// Mitsubishi GX Works2 project: BookEX6_32 Shift_old   PLC: Q13UDV

// global labels: Global
VAR_GLOBAL
  bVar0 AT M5000 : BOOL;
  abArray0 AT M5010 : ARRAY [0..49] OF BOOL;
  sStr0 AT D5000 : STRING[199];
  sStr1 AT D5100 : STRING[199];
  sStr2 AT D5200 : STRING[199];
  sStr3 AT D5300 : STRING[199];
  sStr4 AT D5400 : STRING[199];
  sStr5 AT D5500 : STRING[199];
  sStr6 AT D5600 : STRING[199];
  sStr7 AT D5700 : STRING[199];
  sStr8 AT D5800 : STRING[199];
  sStr9 AT D5900 : STRING[199];
  iVar0 AT D4500 : INT;
  iVar1 AT D4501 : INT;
  iVar2 AT D4502 : INT;
  iVar3 AT D4503 : INT;
  iVar4 AT D4504 : INT;
  iVar5 AT D4505 : INT;
  iVar6 AT D4506 : INT;
  iVar7 AT D4507 : INT;
  iVar8 AT D4508 : INT;
  iVar9 AT D4509 : INT;
  dVar0 AT D4510 : DINT;
  dVar1 AT D4512 : DINT;
  dVar2 AT D4514 : DINT;
  dVar3 AT D4516 : DINT;
  dVar4 AT D4518 : DINT;
  dVar5 AT D4520 : DINT;
  dVar6 AT D4522 : DINT;
  dVar7 AT D4524 : DINT;
  dVar8 AT D4526 : DINT;
  dVar9 AT D4528 : DINT;
  wVar0 AT D4530 : WORD;
  wVar1 AT D4531 : WORD;
  wVar2 AT D4532 : WORD;
  wVar3 AT D4533 : WORD;
  wVar4 AT D4534 : WORD;
  wVar5 AT D4535 : WORD;
  wVar6 AT D4536 : WORD;
  wVar7 AT D4537 : WORD;
  wVar8 AT D4538 : WORD;
  wVar9 AT D4539 : WORD;
  dwVar0 AT D4540 : DWORD;
  dwVar1 AT D4542 : DWORD;
  dwVar2 AT D4544 : DWORD;
  dwVar3 AT D4546 : DWORD;
  dwVar4 AT D4548 : DWORD;
  dwVar5 AT D4550 : DWORD;
  dwVar6 AT D4552 : DWORD;
  dwVar7 AT D4554 : DWORD;
  dwVar8 AT D4556 : DWORD;
  dwVar9 AT D4558 : DWORD;
  fsVar0 AT D4560 : REAL;
  fsVar1 AT D4562 : REAL;
  fsVar2 AT D4564 : REAL;
  fsVar3 AT D4566 : REAL;
  fsVar4 AT D4568 : REAL;
  fsVar5 AT D4570 : REAL;
  fsVar6 AT D4572 : REAL;
  fsVar7 AT D4574 : REAL;
  fsVar8 AT D4576 : REAL;
  fsVar9 AT D4578 : REAL;
  fdVar0 AT D4580 : LREAL;
  tTime0 AT D4620 : TIME;
  tTime1 AT D4622 : TIME;
  tTime2 AT D4624 : TIME;
  tTime3 AT D4626 : TIME;
  tTime4 AT D4628 : TIME;
  tTime5 AT D4630 : TIME;
  tTime6 AT D4632 : TIME;
  tTime7 AT D4634 : TIME;
  tTime8 AT D4636 : TIME;
  tTime9 AT D4638 : TIME;
  tTime10 AT D4640 : TIME;
  bVar1 AT M5001 : BOOL;
  bVar2 AT M5002 : BOOL;
  bVar3 AT M5003 : BOOL;
  bVar4 AT M5004 : BOOL;
  bVar5 AT M5005 : BOOL;
  bVar6 AT M5006 : BOOL;
  bVar7 AT M5007 : BOOL;
  bVar8 AT M5008 : BOOL;
  bVar9 AT M5009 : BOOL;
  abArray1 AT M5060 : ARRAY [0..49] OF BOOL;
  abArray2 AT M5110 : ARRAY [0..49] OF BOOL;
  abArray3 AT M5160 : ARRAY [0..49] OF BOOL;
  abArray4 AT M5210 : ARRAY [0..49] OF BOOL;
  abArray5 AT M5260 : ARRAY [0..49] OF BOOL;
  abArray6 AT M5310 : ARRAY [0..49] OF BOOL;
  abArray7 AT M5360 : ARRAY [0..49] OF BOOL;
  abArray8 AT M5410 : ARRAY [0..49] OF BOOL;
  abArray9 AT M5460 : ARRAY [0..49] OF BOOL;
  fdVar1 AT D4584 : LREAL;
  fdVar2 AT D4588 : LREAL;
  fdVar3 AT D4592 : LREAL;
  fdVar4 AT D4596 : LREAL;
  fdVar5 AT D4600 : LREAL;
  fdVar6 AT D4604 : LREAL;
  fdVar7 AT D4608 : LREAL;
  fdVar8 AT D4612 : LREAL;
  fdVar9 AT D4616 : LREAL;
  afsPen0 AT D2000 : ARRAY [0..499] OF REAL;
  afsPen1 AT D3000 : ARRAY [0..499] OF REAL;
  adwD10 AT D10 : ARRAY [0..9] OF DWORD;
  awLeft AT D10 : ARRAY [0..9] OF WORD;
  awRight AT D20 : ARRAY [0..9] OF WORD;
  awBuffer AT D30 : ARRAY [0..59] OF WORD;
  awDigit AT D100 : ARRAY [0..11,0..9] OF WORD;
  abM10 AT M10 : ARRAY [0..19] OF BOOL;
END_VAR
// user libraries (not included): HMI

FUNCTION BitCount
VAR_INPUT
  w_IN : WORD;
END_VAR
VAR
  wTmp : WORD;
  iCnt : INT;
END_VAR
;
iCnt := 0;
wTmp := w_IN;
WHILE (wTmp AND HFFFF) <> 0 DO
	IF (wTmp  AND 1) <> 0 THEN iCnt := iCnt + 1; END_IF;
	SFR(TRUE, 1, wTmp);
END_WHILE;
BitCount := iCnt;
END_FUNCTION

FUNCTION BitLoadPos
VAR_INPUT
  w_IN : WORD;
END_VAR
VAR
  wInput : WORD;
END_VAR
VAR_INPUT
  b_Val : BOOL;
  i_Pos : INT;
END_VAR
VAR
  wTmp1 : WORD;
  wTmp2 : WORD;
END_VAR
;
wTmp1 := H0001;
wInput := w_IN;
IF b_Val THEN
	SFL(TRUE, i_Pos, wTmp1);
	wTmp2 := wInput OR wTmp1;
ELSE
	SFL(TRUE, i_Pos, wTmp1);
	wTmp2 := wInput AND NOT wTmp1;
END_IF;
BitLoadPos := wTmp2;
END_FUNCTION

FUNCTION BitReset
VAR_INPUT
  w_IN : WORD;
END_VAR
VAR
  wInput : WORD;
END_VAR
VAR_INPUT
  i_Pos : INT;
END_VAR
VAR
  wTmp1 : WORD;
  wTmp2 : WORD;
END_VAR
;
wTmp1 := H0001;
wInput := w_IN;
SFL(TRUE, i_Pos, wTmp1);
wTmp2 := wInput AND NOT wTmp1;
BitReset := wTmp2;
END_FUNCTION

FUNCTION BitSet
VAR_INPUT
  w_IN : WORD;
END_VAR
VAR
  wInput : WORD;
END_VAR
VAR_INPUT
  i_Pos : INT;
END_VAR
VAR
  wTmp1 : WORD;
  wTmp2 : WORD;
END_VAR
;
wTmp1 := H0001;
wInput := w_IN;
SFL(TRUE, i_Pos, wTmp1);
wTmp2 := wInput OR wTmp1;
BitSet := wTmp2;
END_FUNCTION

FUNCTION BitToggle
VAR_INPUT
  w_IN : WORD;
  i_Pos : INT;
END_VAR
VAR
  wInput : WORD;
  wTmp1 : WORD;
  wTmp2 : WORD;
END_VAR
;
wTmp1 := H0001;
wInput := w_IN;
SFL(TRUE, i_Pos, wTmp1);
wTmp2 := wInput XOR wTmp1;
BitToggle := wTmp2;
END_FUNCTION

FUNCTION_BLOCK EBIncDec
VAR_INPUT
  i_Old : INT;
END_VAR
VAR_OUTPUT
  b_ChgUp : BOOL;
END_VAR
VAR_INPUT
  b_Inc : BOOL;
END_VAR
VAR
  ix : INT;
END_VAR
VAR_OUTPUT
  i_New : INT;
END_VAR
VAR_INPUT
  b_Dec : BOOL;
END_VAR
VAR_OUTPUT
  b_ChgDw : BOOL;
END_VAR
;
IF NOT b_Inc AND NOT b_Dec THEN
	RETURN;
END_IF;
IF b_Inc THEN
	IF  (i_Old = 9) OR (i_Old = 0) THEN
		b_ChgUp := FALSE;
	ELSE
		i_New := i_Old + 1;
		b_ChgUp := TRUE;
		FOR ix := 0 TO 9 DO 
			awBuffer[ix+20] := awDigit[10, ix];
			awBuffer[ix+50] := awDigit[i_New, ix];
		END_FOR;
	END_IF;
ELSIF b_Dec THEN
	IF  (i_Old = 1) OR (i_Old = 0) THEN
		b_ChgDw := FALSE;
	ELSE
		i_New := i_Old - 1;
		b_ChgDw := TRUE;
		FOR ix := 0 TO 9 DO 
			awBuffer[ix+0] := awDigit[11, ix];
			awBuffer[ix+30] := awDigit[i_New, ix];
		END_FOR;
	END_IF;
END_IF;
END_FUNCTION_BLOCK

FUNCTION_BLOCK EBScroll
VAR_INPUT
  b_EN : BOOL;
  b_Up : BOOL;
  b_Dw : BOOL;
END_VAR
VAR_OUTPUT
  b_Ing : BOOL;
  b_Comp : BOOL;
END_VAR
VAR
  ix : INT;
  iCnt : INT;
END_VAR
VAR_IN_OUT
  i_Old : INT;
  i_New : INT;
END_VAR
VAR
  fbTimer : TON;
END_VAR
;
IF NOT b_EN THEN
	iCnt := 0;
	b_Ing := FALSE;
	b_Comp := FALSE;
	fbTimer(IN:=FALSE);
	RETURN;
END_IF;

IF b_Up THEN
	CASE iCnt OF 
		0 : 	FOR ix := 0 TO 9 DO 
					awBuffer[ix+10] := 0;
					awBuffer[ix+40] := awDigit[i_Old, ix];
				END_FOR;
				b_Comp := FALSE;
				b_Ing := TRUE;
				iCnt := iCnt + 1;
		1..10 : 
				fbTimer(IN := TRUE , PT:=T#500ms);
				IF fbTimer.Q THEN
					fbTimer(IN:=FALSE);
					iCnt := iCnt+1;
					SFTWR(TRUE, 30, 1, awBuffer[0] );
					SFTWR(TRUE, 30, 1, awBuffer[30] );
				END_IF;
		11..14 : 
				fbTimer(IN := TRUE , PT:=T#500ms);
				IF fbTimer.Q THEN
					fbTimer(IN:=FALSE);
					iCnt := iCnt+1;
					SFTWR(TRUE, 30, 1, awBuffer[0] );
				END_IF;
		15 :		
				b_Comp := TRUE;
				i_Old := i_New;
				b_Ing := FALSE;
				iCnt := 0;
	END_CASE;
ELSIF b_Dw THEN
	CASE iCnt OF 
		0 : 	FOR ix := 0 TO 9 DO 
					awBuffer[ix+10] := 0;
					awBuffer[ix+40] := awDigit[i_Old, ix];
				END_FOR;
				b_Comp := FALSE;
				b_Ing := TRUE;
				iCnt := iCnt + 1;
		1..10 : 
				fbTimer(IN := TRUE , PT:=T#500ms);
				IF fbTimer.Q THEN
					fbTimer(IN:=FALSE);
					iCnt := iCnt+1;
					SFTWL(TRUE, 30, 1, awBuffer[0] );
					SFTWL(TRUE, 30, 1, awBuffer[30] );
				END_IF;
		11..15 : 
				fbTimer(IN := TRUE , PT:=T#500ms);
				IF fbTimer.Q THEN
					fbTimer(IN:=FALSE);
					iCnt := iCnt+1;
					SFTWL(TRUE, 30, 1, awBuffer[0] );
				END_IF;
		16 :		
				b_Comp := TRUE;
				i_Old := i_New;
				b_Ing := FALSE;
				iCnt := 0;
	END_CASE;	
ELSE
	iCnt := 0;
	b_Ing := FALSE;
	b_Comp := FALSE;
	FOR ix := 0 TO 9 DO 
		awBuffer[ix+10] := 0;
		awBuffer[ix+40] := awDigit[i_Old, ix];
	END_FOR;
END_IF;

FOR ix := 0 TO 9 DO 
		awLeft[ix] := awBuffer[ix+10];
		awRight[ix] := awBuffer[ix+40];
END_FOR;
END_FUNCTION_BLOCK

FUNCTION_BLOCK EBScroll2
VAR_INPUT
  b_EN : BOOL;
  b_Up : BOOL;
  b_Dw : BOOL;
END_VAR
VAR_OUTPUT
  b_Ing : BOOL;
  b_Comp : BOOL;
END_VAR
VAR
  ix : INT;
  iCnt : INT;
END_VAR
VAR_IN_OUT
  i_Old : INT;
  i_New : INT;
END_VAR
VAR
  fbTimer : TON;
  dwTemp1 : DWORD;
  dwTemp2 : DWORD;
  dwTemp3 : DWORD;
  dwTemp4 : DWORD;
  dwTemp5 : DWORD;
  iy : INT;
END_VAR
;
IF NOT b_EN THEN
	iCnt := 0;
	b_Ing := FALSE;
	b_Comp := FALSE;
	fbTimer(IN:=FALSE);
	RETURN;
END_IF;

IF b_Up THEN
	CASE iCnt OF 
		0 : 	FOR ix := 0 TO 9 DO 
					awBuffer[ix+10] := 0;
					awBuffer[ix+40] := awDigit[i_Old, ix];
				END_FOR;
				b_Comp := FALSE;
				b_Ing := TRUE;
				iCnt := iCnt + 1;
		1..16 : 
				fbTimer(IN := TRUE , PT:=T#500ms);
				IF fbTimer.Q THEN
					fbTimer(IN:=FALSE);
					iCnt := iCnt+1;
					FOR iy := 0 TO 9 DO
						dwTemp1 			:= WORD_TO_DWORD(awBuffer[iy+40]) AND H000000FF;
						dwTemp2 			:= SHL( WORD_TO_DWORD(awBuffer[iy+10]), 8) AND H0000FF00;
						dwTemp3 			:= SHL( WORD_TO_DWORD(awBuffer[iy+50]), 16) AND H00FF0000;
						dwTemp4 			:= SHL( WORD_TO_DWORD(awBuffer[iy+20]), 24) AND HFF000000;
						dwTemp5 			:= dwTemp1 OR dwTemp2 OR dwTemp3 OR dwTemp4;
						dwTemp5 			:= SHR(dwTemp5, 1);
						awBuffer[iy+40] 	:= DWORD_TO_WORD(dwTemp5 AND H000000FF);
						awBuffer[iy+10] 	:= DWORD_TO_WORD(SHR(dwTemp5, 8) AND H000000FF);
						awBuffer[iy+50] 	:= DWORD_TO_WORD(SHR(dwTemp5, 16) AND H000000FF);
						awBuffer[iy+20]	:= DWORD_TO_WORD(SHR(dwTemp5, 24) AND H000000FF);
					END_FOR;
				END_IF;
		17 :		
				b_Comp := TRUE;
				i_Old := i_New;
				b_Ing := FALSE;
				iCnt := 0;
	END_CASE;
ELSIF b_Dw THEN
	CASE iCnt OF 
		0 : 	FOR ix := 0 TO 9 DO 
					awBuffer[ix+10] := 0;
					awBuffer[ix+40] := awDigit[i_Old, ix];
				END_FOR;
				b_Comp := FALSE;
				b_Ing := TRUE;
				iCnt := iCnt + 1;
		1..16 : 
				fbTimer(IN := TRUE , PT:=T#500ms);
				IF fbTimer.Q THEN
					fbTimer(IN:=FALSE);
					iCnt := iCnt+1;
					FOR iy := 0 TO 9 DO
						dwTemp1 			:= WORD_TO_DWORD(awBuffer[iy+30]) AND H000000FF;
						dwTemp2 			:= SHL( WORD_TO_DWORD(awBuffer[iy]), 8) AND H0000FF00;
						dwTemp3 			:= SHL( WORD_TO_DWORD(awBuffer[iy+40]), 16) AND H00FF0000;
						dwTemp4 			:= SHL( WORD_TO_DWORD(awBuffer[iy+10]), 24) AND HFF000000;
						dwTemp5 			:= dwTemp1 OR dwTemp2 OR dwTemp3 OR dwTemp4;
						dwTemp5 			:= SHL(dwTemp5, 1);
						awBuffer[iy+30] 	:= DWORD_TO_WORD(dwTemp5 AND H000000FF);
						awBuffer[iy] 		:= DWORD_TO_WORD(SHR(dwTemp5, 8) AND H000000FF);
						awBuffer[iy+40] 	:= DWORD_TO_WORD(SHR(dwTemp5, 16) AND H000000FF);
						awBuffer[iy+10]	:= DWORD_TO_WORD(SHR(dwTemp5, 24) AND H000000FF);
					END_FOR;
				END_IF;
		17 :		
				b_Comp := TRUE;
				i_Old := i_New;
				b_Ing := FALSE;
				iCnt := 0;
	END_CASE;	
ELSE
	iCnt := 0;
	b_Ing := FALSE;
	b_Comp := FALSE;
	FOR ix := 0 TO 9 DO 
		awBuffer[ix+10] := 0;
		awBuffer[ix+40] := awDigit[i_Old, ix];
	END_FOR;
END_IF;

FOR ix := 0 TO 9 DO 
		awLeft[ix] := awBuffer[ix+10];
		awRight[ix] := awBuffer[ix+40];
END_FOR;
END_FUNCTION_BLOCK

PROGRAM ExBSFR
(* structured ladder/FBD written out as ST: instructions are called as NAME(EN, inputs, outputs); _pN, _eN, _tN stand for wires *)
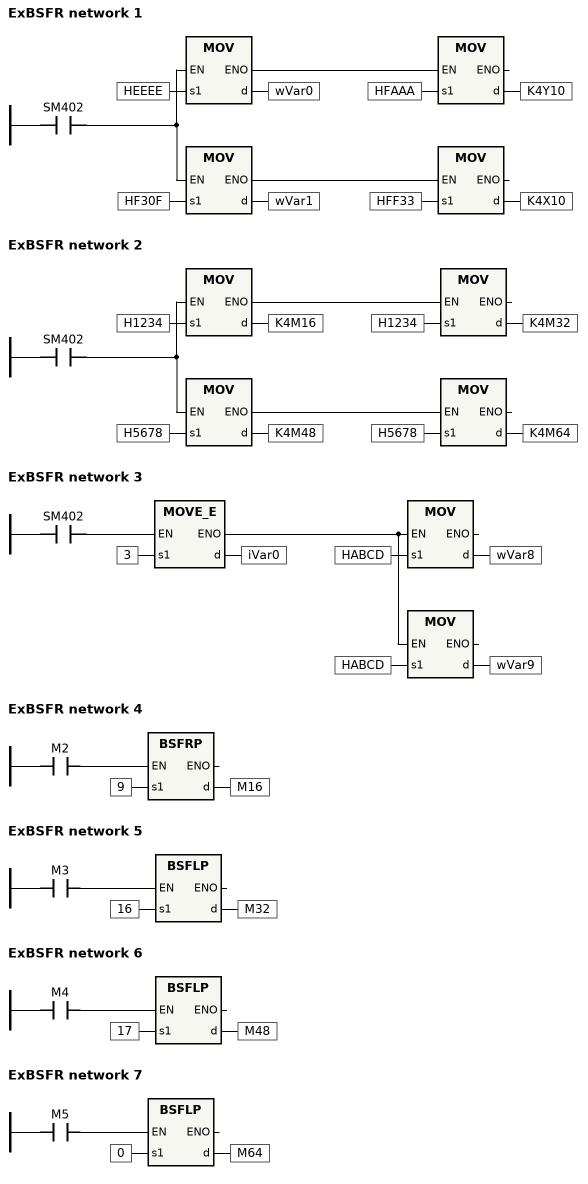
(* network 1 *)
_e1 := MOV(SM402, HEEEE, wVar0);
MOV(_e1, HFAAA, K4Y10);
_e2 := MOV(SM402, HF30F, wVar1);
MOV(_e2, HFF33, K4X10);
(* network 2 *)
_e1 := MOV(SM402, H1234, K4M16);
MOV(_e1, H1234, K4M32);
_e2 := MOV(SM402, H5678, K4M48);
MOV(_e2, H5678, K4M64);
(* network 3 *)
_e1 := MOVE_E(SM402, 3, iVar0);
MOV(_e1, HABCD, wVar8);
MOV(_e1, HABCD, wVar9);
(* network 4 *)
BSFRP(M2, 9, M16);
(* network 5 *)
BSFLP(M3, 16, M32);
(* network 6 *)
BSFLP(M4, 17, M48);
(* network 7 *)
BSFLP(M5, 0, M64);
END_PROGRAM

PROGRAM ExDisplay
VAR
  Mov8WORD_1 : Mov8WORD;
  Mov8WORD_2 : Mov8WORD;
  Mov8WORD_3 : Mov8WORD;
  Mov8WORD_4 : Mov8WORD;
  Mov8WORD_5 : Mov8WORD;
  Mov8WORD_6 : Mov8WORD;
  Mov8WORD_7 : Mov8WORD;
  Mov8WORD_8 : Mov8WORD;
  Mov8WORD_9 : Mov8WORD;
  Mov8WORD_10 : Mov8WORD;
  Mov8WORD_11 : Mov8WORD;
  Mov8WORD_12 : Mov8WORD;
  Mov8WORD_13 : Mov8WORD;
  Mov8WORD_14 : Mov8WORD;
  Mov8WORD_15 : Mov8WORD;
  OldIdx : INT;
  NewIdx : INT;
  bDwFlag : BOOL;
  bUpFlag : BOOL;
  EBScroll_1 : EBScroll;
  bScroll : BOOL;
  bStop : BOOL;
  EBIncDec_1 : EBIncDec;
END_VAR
(* structured ladder/FBD written out as ST: instructions are called as NAME(EN, inputs, outputs); _pN, _eN, _tN stand for wires *)
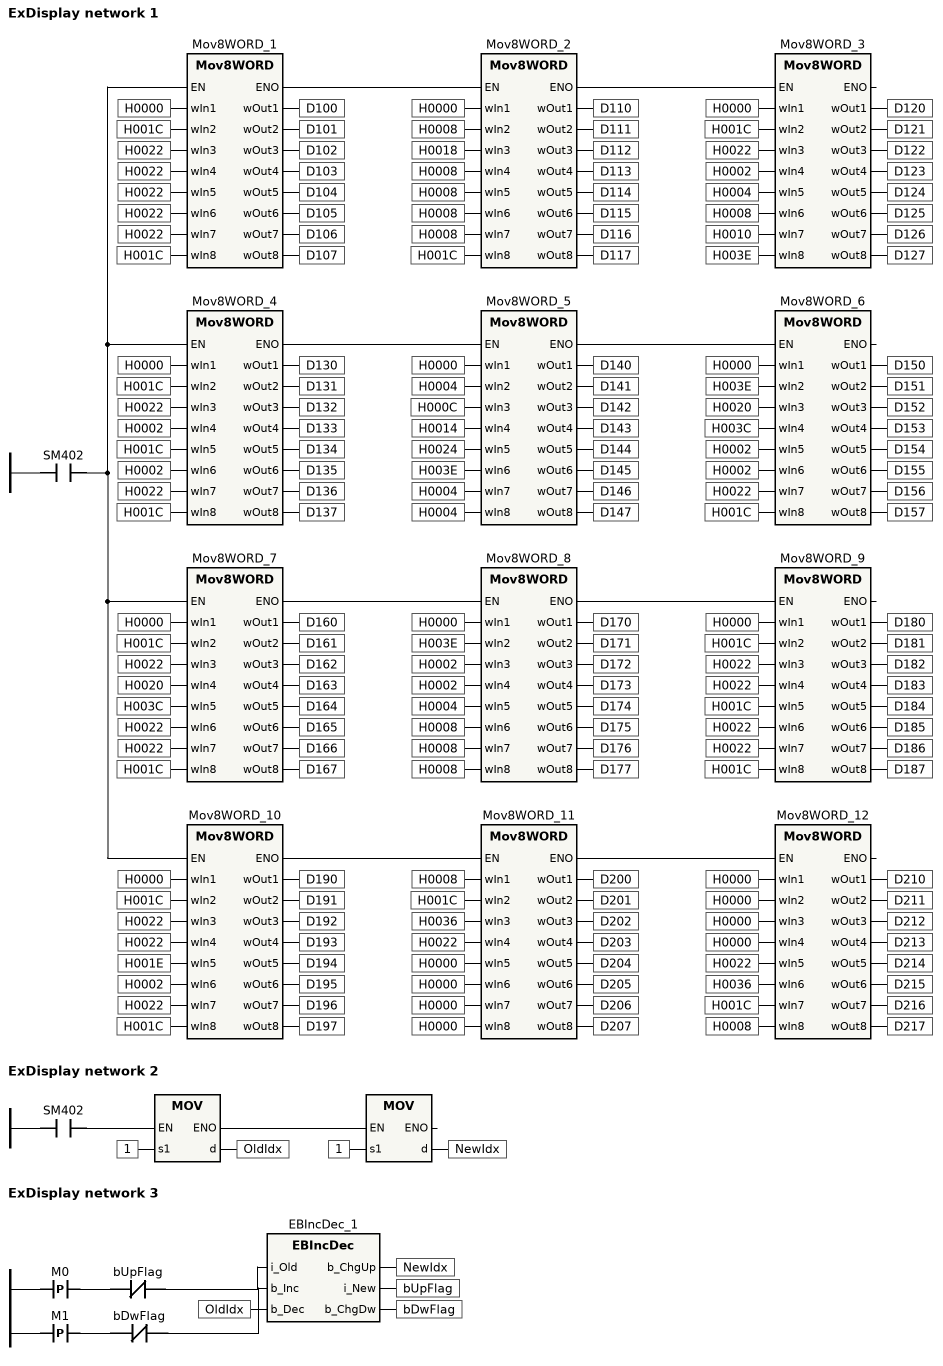
(* network 1 *)
Mov8WORD_1(EN := SM402, wIn1 := H0000, wIn2 := H001C, wIn3 := H0022, wIn4 := H0022, wIn5 := H0022, wIn6 := H0022, wIn7 := H0022, wIn8 := H001C, wOut1 => D100, wOut2 => D101, wOut3 => D102, wOut4 => D103, wOut5 => D104, wOut6 => D105, wOut7 => D106, wOut8 => D107);
Mov8WORD_2(EN := Mov8WORD_1.ENO, wIn1 := H0000, wIn2 := H0008, wIn3 := H0018, wIn4 := H0008, wIn5 := H0008, wIn6 := H0008, wIn7 := H0008, wIn8 := H001C, wOut1 => D110, wOut2 => D111, wOut3 => D112, wOut4 => D113, wOut5 => D114, wOut6 => D115, wOut7 => D116, wOut8 => D117);
Mov8WORD_3(EN := Mov8WORD_2.ENO, wIn1 := H0000, wIn2 := H001C, wIn3 := H0022, wIn4 := H0002, wIn5 := H0004, wIn6 := H0008, wIn7 := H0010, wIn8 := H003E, wOut1 => D120, wOut2 => D121, wOut3 => D122, wOut4 => D123, wOut5 => D124, wOut6 => D125, wOut7 => D126, wOut8 => D127);
Mov8WORD_4(EN := SM402, wIn1 := H0000, wIn2 := H001C, wIn3 := H0022, wIn4 := H0002, wIn5 := H001C, wIn6 := H0002, wIn7 := H0022, wIn8 := H001C, wOut1 => D130, wOut2 => D131, wOut3 => D132, wOut4 => D133, wOut5 => D134, wOut6 => D135, wOut7 => D136, wOut8 => D137);
Mov8WORD_5(EN := Mov8WORD_4.ENO, wIn1 := H0000, wIn2 := H0004, wIn3 := H000C, wIn4 := H0014, wIn5 := H0024, wIn6 := H003E, wIn7 := H0004, wIn8 := H0004, wOut1 => D140, wOut2 => D141, wOut3 => D142, wOut4 => D143, wOut5 => D144, wOut6 => D145, wOut7 => D146, wOut8 => D147);
Mov8WORD_6(EN := Mov8WORD_5.ENO, wIn1 := H0000, wIn2 := H003E, wIn3 := H0020, wIn4 := H003C, wIn5 := H0002, wIn6 := H0002, wIn7 := H0022, wIn8 := H001C, wOut1 => D150, wOut2 => D151, wOut3 => D152, wOut4 => D153, wOut5 => D154, wOut6 => D155, wOut7 => D156, wOut8 => D157);
Mov8WORD_7(EN := SM402, wIn1 := H0000, wIn2 := H001C, wIn3 := H0022, wIn4 := H0020, wIn5 := H003C, wIn6 := H0022, wIn7 := H0022, wIn8 := H001C, wOut1 => D160, wOut2 => D161, wOut3 => D162, wOut4 => D163, wOut5 => D164, wOut6 => D165, wOut7 => D166, wOut8 => D167);
Mov8WORD_8(EN := Mov8WORD_7.ENO, wIn1 := H0000, wIn2 := H003E, wIn3 := H0002, wIn4 := H0002, wIn5 := H0004, wIn6 := H0008, wIn7 := H0008, wIn8 := H0008, wOut1 => D170, wOut2 => D171, wOut3 => D172, wOut4 => D173, wOut5 => D174, wOut6 => D175, wOut7 => D176, wOut8 => D177);
Mov8WORD_9(EN := Mov8WORD_8.ENO, wIn1 := H0000, wIn2 := H001C, wIn3 := H0022, wIn4 := H0022, wIn5 := H001C, wIn6 := H0022, wIn7 := H0022, wIn8 := H001C, wOut1 => D180, wOut2 => D181, wOut3 => D182, wOut4 => D183, wOut5 => D184, wOut6 => D185, wOut7 => D186, wOut8 => D187);
Mov8WORD_10(EN := SM402, wIn1 := H0000, wIn2 := H001C, wIn3 := H0022, wIn4 := H0022, wIn5 := H001E, wIn6 := H0002, wIn7 := H0022, wIn8 := H001C, wOut1 => D190, wOut2 => D191, wOut3 => D192, wOut4 => D193, wOut5 => D194, wOut6 => D195, wOut7 => D196, wOut8 => D197);
Mov8WORD_11(EN := Mov8WORD_10.ENO, wIn1 := H0008, wIn2 := H001C, wIn3 := H0036, wIn4 := H0022, wIn5 := H0000, wIn6 := H0000, wIn7 := H0000, wIn8 := H0000, wOut1 => D200, wOut2 => D201, wOut3 => D202, wOut4 => D203, wOut5 => D204, wOut6 => D205, wOut7 => D206, wOut8 => D207);
Mov8WORD_12(EN := Mov8WORD_11.ENO, wIn1 := H0000, wIn2 := H0000, wIn3 := H0000, wIn4 := H0000, wIn5 := H0022, wIn6 := H0036, wIn7 := H001C, wIn8 := H0008, wOut1 => D210, wOut2 => D211, wOut3 => D212, wOut4 => D213, wOut5 => D214, wOut6 => D215, wOut7 => D216, wOut8 => D217);
(* network 2 *)
_e1 := MOV(SM402, 1, OldIdx);
MOV(_e1, 1, NewIdx);
(* network 3 *)
EBIncDec_1(i_Old := LDP(TRUE, M0) AND NOT bUpFlag, b_Inc := LDP(TRUE, M1) AND NOT bDwFlag, b_Dec := OldIdx, b_ChgUp => NewIdx, i_New => bUpFlag, b_ChgDw => bDwFlag);
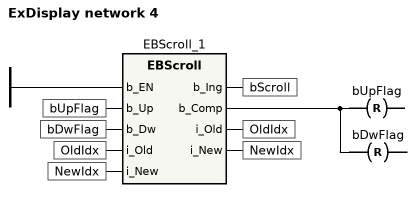
(* network 4 *)
EBScroll_1(b_EN := TRUE, b_Up := bUpFlag, b_Dw := bDwFlag, i_Old := OldIdx, i_New := NewIdx, b_Ing => bScroll);
RST(EBScroll_1.b_Comp, bUpFlag);
OldIdx := EBScroll_1.i_Old;
RST(EBScroll_1.b_Comp, bDwFlag);
NewIdx := EBScroll_1.i_New;
END_PROGRAM

PROGRAM ExDisplay2
VAR
  Mov8WORD_1 : Mov8WORD;
  Mov8WORD_2 : Mov8WORD;
  Mov8WORD_3 : Mov8WORD;
  Mov8WORD_4 : Mov8WORD;
  Mov8WORD_5 : Mov8WORD;
  Mov8WORD_6 : Mov8WORD;
  Mov8WORD_7 : Mov8WORD;
  Mov8WORD_8 : Mov8WORD;
  Mov8WORD_9 : Mov8WORD;
  Mov8WORD_10 : Mov8WORD;
  Mov8WORD_11 : Mov8WORD;
  Mov8WORD_12 : Mov8WORD;
  Mov8WORD_13 : Mov8WORD;
  Mov8WORD_14 : Mov8WORD;
  Mov8WORD_15 : Mov8WORD;
  OldIdx : INT;
  NewIdx : INT;
  bDwFlag : BOOL;
  bUpFlag : BOOL;
  bScroll : BOOL;
  bStop : BOOL;
  EBScroll_1 : EBScroll2;
  EBIncDec_1 : EBIncDec;
END_VAR
(* structured ladder/FBD written out as ST: instructions are called as NAME(EN, inputs, outputs); _pN, _eN, _tN stand for wires *)
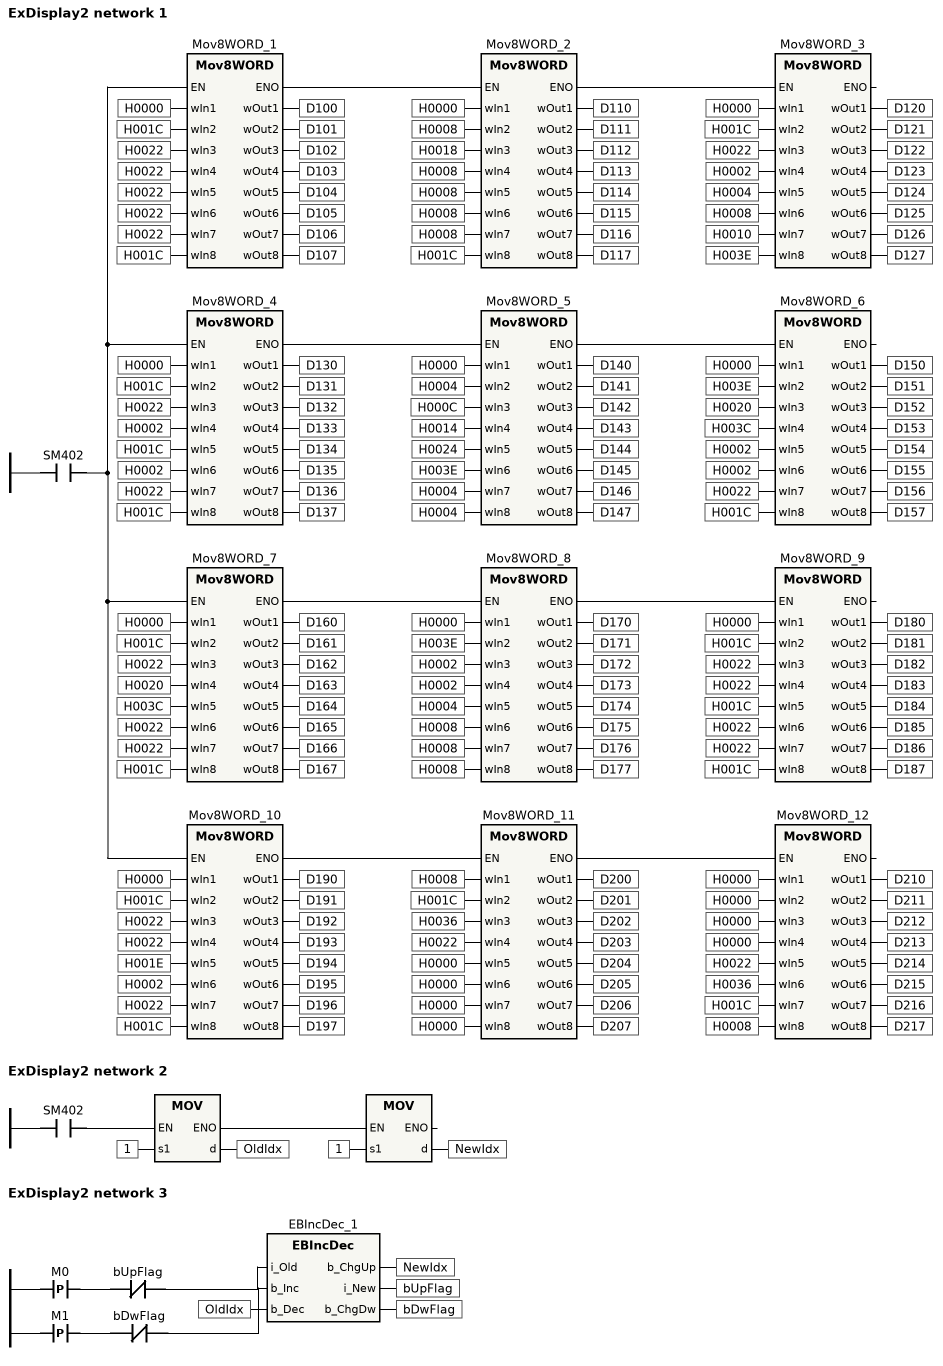
(* network 1 *)
Mov8WORD_1(EN := SM402, wIn1 := H0000, wIn2 := H001C, wIn3 := H0022, wIn4 := H0022, wIn5 := H0022, wIn6 := H0022, wIn7 := H0022, wIn8 := H001C, wOut1 => D100, wOut2 => D101, wOut3 => D102, wOut4 => D103, wOut5 => D104, wOut6 => D105, wOut7 => D106, wOut8 => D107);
Mov8WORD_2(EN := Mov8WORD_1.ENO, wIn1 := H0000, wIn2 := H0008, wIn3 := H0018, wIn4 := H0008, wIn5 := H0008, wIn6 := H0008, wIn7 := H0008, wIn8 := H001C, wOut1 => D110, wOut2 => D111, wOut3 => D112, wOut4 => D113, wOut5 => D114, wOut6 => D115, wOut7 => D116, wOut8 => D117);
Mov8WORD_3(EN := Mov8WORD_2.ENO, wIn1 := H0000, wIn2 := H001C, wIn3 := H0022, wIn4 := H0002, wIn5 := H0004, wIn6 := H0008, wIn7 := H0010, wIn8 := H003E, wOut1 => D120, wOut2 => D121, wOut3 => D122, wOut4 => D123, wOut5 => D124, wOut6 => D125, wOut7 => D126, wOut8 => D127);
Mov8WORD_4(EN := SM402, wIn1 := H0000, wIn2 := H001C, wIn3 := H0022, wIn4 := H0002, wIn5 := H001C, wIn6 := H0002, wIn7 := H0022, wIn8 := H001C, wOut1 => D130, wOut2 => D131, wOut3 => D132, wOut4 => D133, wOut5 => D134, wOut6 => D135, wOut7 => D136, wOut8 => D137);
Mov8WORD_5(EN := Mov8WORD_4.ENO, wIn1 := H0000, wIn2 := H0004, wIn3 := H000C, wIn4 := H0014, wIn5 := H0024, wIn6 := H003E, wIn7 := H0004, wIn8 := H0004, wOut1 => D140, wOut2 => D141, wOut3 => D142, wOut4 => D143, wOut5 => D144, wOut6 => D145, wOut7 => D146, wOut8 => D147);
Mov8WORD_6(EN := Mov8WORD_5.ENO, wIn1 := H0000, wIn2 := H003E, wIn3 := H0020, wIn4 := H003C, wIn5 := H0002, wIn6 := H0002, wIn7 := H0022, wIn8 := H001C, wOut1 => D150, wOut2 => D151, wOut3 => D152, wOut4 => D153, wOut5 => D154, wOut6 => D155, wOut7 => D156, wOut8 => D157);
Mov8WORD_7(EN := SM402, wIn1 := H0000, wIn2 := H001C, wIn3 := H0022, wIn4 := H0020, wIn5 := H003C, wIn6 := H0022, wIn7 := H0022, wIn8 := H001C, wOut1 => D160, wOut2 => D161, wOut3 => D162, wOut4 => D163, wOut5 => D164, wOut6 => D165, wOut7 => D166, wOut8 => D167);
Mov8WORD_8(EN := Mov8WORD_7.ENO, wIn1 := H0000, wIn2 := H003E, wIn3 := H0002, wIn4 := H0002, wIn5 := H0004, wIn6 := H0008, wIn7 := H0008, wIn8 := H0008, wOut1 => D170, wOut2 => D171, wOut3 => D172, wOut4 => D173, wOut5 => D174, wOut6 => D175, wOut7 => D176, wOut8 => D177);
Mov8WORD_9(EN := Mov8WORD_8.ENO, wIn1 := H0000, wIn2 := H001C, wIn3 := H0022, wIn4 := H0022, wIn5 := H001C, wIn6 := H0022, wIn7 := H0022, wIn8 := H001C, wOut1 => D180, wOut2 => D181, wOut3 => D182, wOut4 => D183, wOut5 => D184, wOut6 => D185, wOut7 => D186, wOut8 => D187);
Mov8WORD_10(EN := SM402, wIn1 := H0000, wIn2 := H001C, wIn3 := H0022, wIn4 := H0022, wIn5 := H001E, wIn6 := H0002, wIn7 := H0022, wIn8 := H001C, wOut1 => D190, wOut2 => D191, wOut3 => D192, wOut4 => D193, wOut5 => D194, wOut6 => D195, wOut7 => D196, wOut8 => D197);
Mov8WORD_11(EN := Mov8WORD_10.ENO, wIn1 := H0008, wIn2 := H001C, wIn3 := H0036, wIn4 := H0022, wIn5 := H0000, wIn6 := H0000, wIn7 := H0000, wIn8 := H0000, wOut1 => D200, wOut2 => D201, wOut3 => D202, wOut4 => D203, wOut5 => D204, wOut6 => D205, wOut7 => D206, wOut8 => D207);
Mov8WORD_12(EN := Mov8WORD_11.ENO, wIn1 := H0000, wIn2 := H0000, wIn3 := H0000, wIn4 := H0000, wIn5 := H0022, wIn6 := H0036, wIn7 := H001C, wIn8 := H0008, wOut1 => D210, wOut2 => D211, wOut3 => D212, wOut4 => D213, wOut5 => D214, wOut6 => D215, wOut7 => D216, wOut8 => D217);
(* network 2 *)
_e1 := MOV(SM402, 1, OldIdx);
MOV(_e1, 1, NewIdx);
(* network 3 *)
EBIncDec_1(i_Old := LDP(TRUE, M0) AND NOT bUpFlag, b_Inc := LDP(TRUE, M1) AND NOT bDwFlag, b_Dec := OldIdx, b_ChgUp => NewIdx, i_New => bUpFlag, b_ChgDw => bDwFlag);
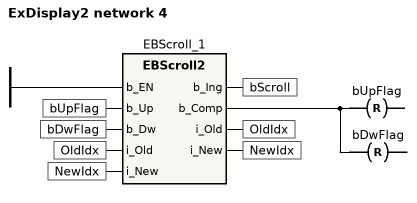
(* network 4 *)
EBScroll_1(b_EN := TRUE, b_Up := bUpFlag, b_Dw := bDwFlag, i_Old := OldIdx, i_New := NewIdx, b_Ing => bScroll);
RST(EBScroll_1.b_Comp, bUpFlag);
OldIdx := EBScroll_1.i_Old;
RST(EBScroll_1.b_Comp, bDwFlag);
NewIdx := EBScroll_1.i_New;
END_PROGRAM

PROGRAM ExDSFR
VAR
  Mov4WORD_1 : Mov4WORD;
  Mov8INT_1 : Mov8INT;
  Mov8INT_2 : Mov8INT;
END_VAR
(* structured ladder/FBD written out as ST: instructions are called as NAME(EN, inputs, outputs); _pN, _eN, _tN stand for wires *)
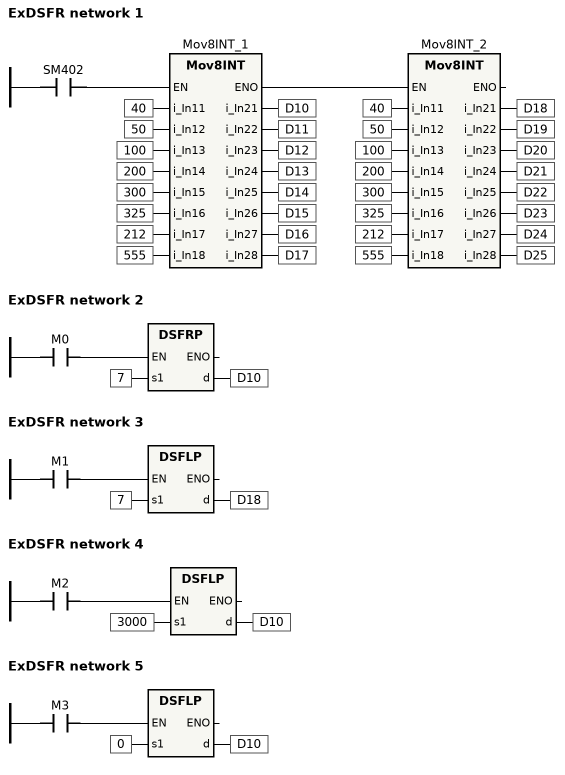
(* network 1 *)
Mov8INT_1(EN := SM402, i_In11 := 40, i_In12 := 50, i_In13 := 100, i_In14 := 200, i_In15 := 300, i_In16 := 325, i_In17 := 212, i_In18 := 555, i_In21 => D10, i_In22 => D11, i_In23 => D12, i_In24 => D13, i_In25 => D14, i_In26 => D15, i_In27 => D16, i_In28 => D17);
Mov8INT_2(EN := Mov8INT_1.ENO, i_In11 := 40, i_In12 := 50, i_In13 := 100, i_In14 := 200, i_In15 := 300, i_In16 := 325, i_In17 := 212, i_In18 := 555, i_In21 => D18, i_In22 => D19, i_In23 => D20, i_In24 => D21, i_In25 => D22, i_In26 => D23, i_In27 => D24, i_In28 => D25);
(* network 2 *)
DSFRP(M0, 7, D10);
(* network 3 *)
DSFLP(M1, 7, D18);
(* network 4 *)
DSFLP(M2, 3000, D10);
(* network 5 *)
DSFLP(M3, 0, D10);
END_PROGRAM

PROGRAM ExLib
(* structured ladder/FBD written out as ST: instructions are called as NAME(EN, inputs, outputs); _pN, _eN, _tN stand for wires *)
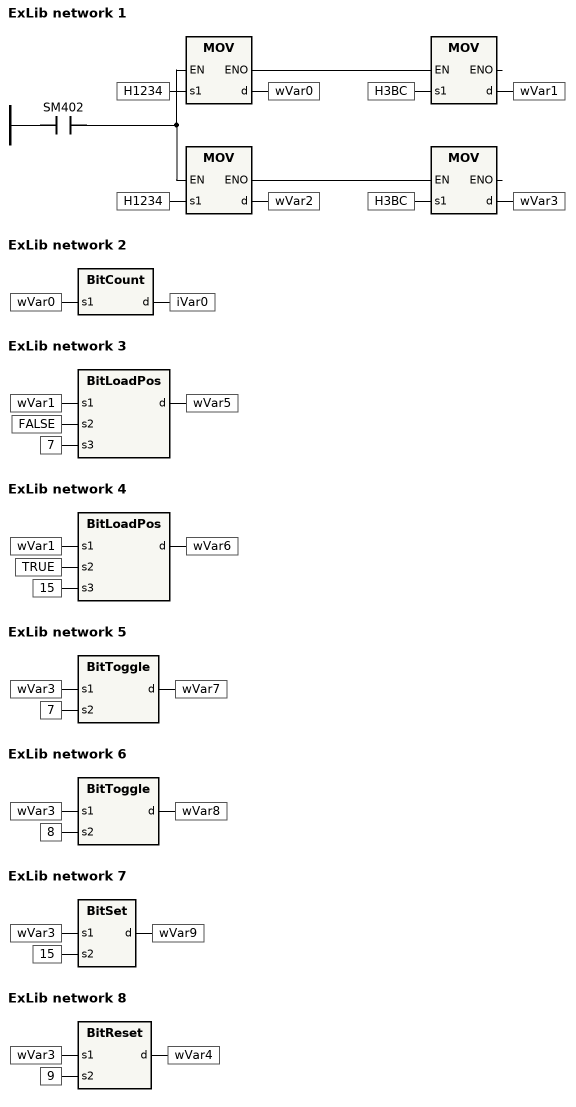
(* network 1 *)
_e1 := MOV(SM402, H1234, wVar0);
MOV(_e1, H3BC, wVar1);
_e2 := MOV(SM402, H1234, wVar2);
MOV(_e2, H3BC, wVar3);
(* network 2 *)
iVar0 := BitCount(wVar0);
(* network 3 *)
wVar5 := BitLoadPos(wVar1, FALSE, 7);
(* network 4 *)
wVar6 := BitLoadPos(wVar1, TRUE, 15);
(* network 5 *)
wVar7 := BitToggle(wVar3, 7);
(* network 6 *)
wVar8 := BitToggle(wVar3, 8);
(* network 7 *)
wVar9 := BitSet(wVar3, 15);
(* network 8 *)
wVar4 := BitReset(wVar3, 9);
END_PROGRAM

PROGRAM ExSFR
(* structured ladder/FBD written out as ST: instructions are called as NAME(EN, inputs, outputs); _pN, _eN, _tN stand for wires *)
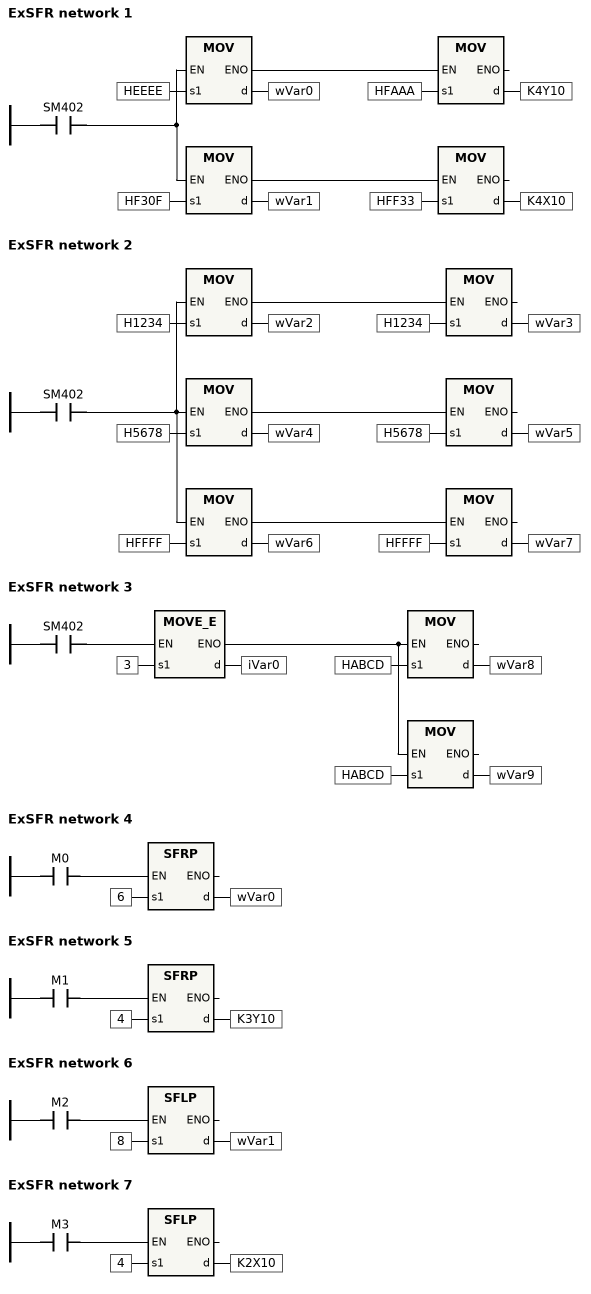
(* network 1 *)
_e1 := MOV(SM402, HEEEE, wVar0);
MOV(_e1, HFAAA, K4Y10);
_e2 := MOV(SM402, HF30F, wVar1);
MOV(_e2, HFF33, K4X10);
(* network 2 *)
_e1 := MOV(SM402, H1234, wVar2);
MOV(_e1, H1234, wVar3);
_e2 := MOV(SM402, H5678, wVar4);
MOV(_e2, H5678, wVar5);
_e3 := MOV(SM402, HFFFF, wVar6);
MOV(_e3, HFFFF, wVar7);
(* network 3 *)
_e1 := MOVE_E(SM402, 3, iVar0);
MOV(_e1, HABCD, wVar8);
MOV(_e1, HABCD, wVar9);
(* network 4 *)
SFRP(M0, 6, wVar0);
(* network 5 *)
SFRP(M1, 4, K3Y10);
(* network 6 *)
SFLP(M2, 8, wVar1);
(* network 7 *)
SFLP(M3, 4, K2X10);
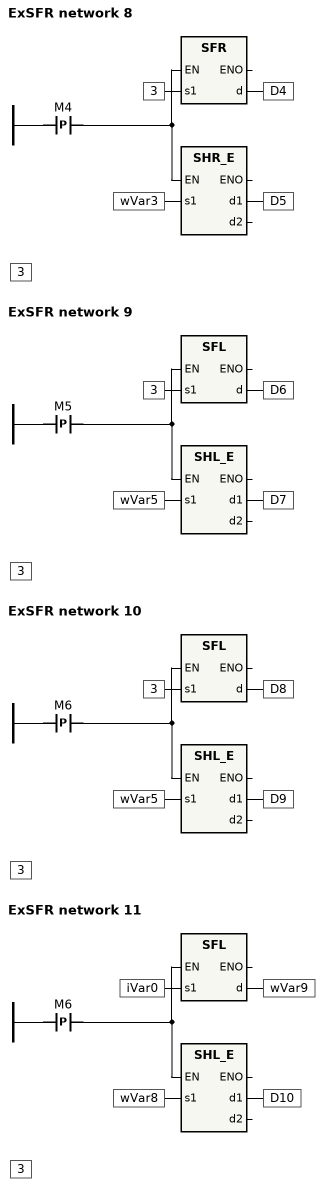
(* network 8 *)
_p1 := LDP(TRUE, M4);
SFR(_p1, 3, D4);
SHR_E(_p1, wVar3, D5, _open);
(* not connected to any output: 3 *)
(* network 9 *)
_p1 := LDP(TRUE, M5);
SFL(_p1, 3, D6);
SHL_E(_p1, wVar5, D7, _open);
(* not connected to any output: 3 *)
(* network 10 *)
_p1 := LDP(TRUE, M6);
SFL(_p1, 3, D8);
SHL_E(_p1, wVar5, D9, _open);
(* not connected to any output: 3 *)
(* network 11 *)
_p1 := LDP(TRUE, M6);
SFL(_p1, iVar0, wVar9);
SHL_E(_p1, wVar8, D10, _open);
(* not connected to any output: 3 *)
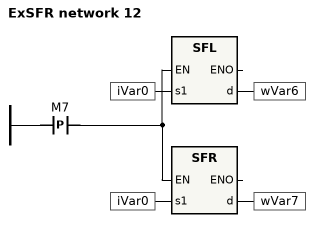
(* network 12 *)
_p1 := LDP(TRUE, M7);
SFL(_p1, iVar0, wVar6);
SFR(_p1, iVar0, wVar7);
END_PROGRAM

PROGRAM ExSFTBR
(* structured ladder/FBD written out as ST: instructions are called as NAME(EN, inputs, outputs); _pN, _eN, _tN stand for wires *)
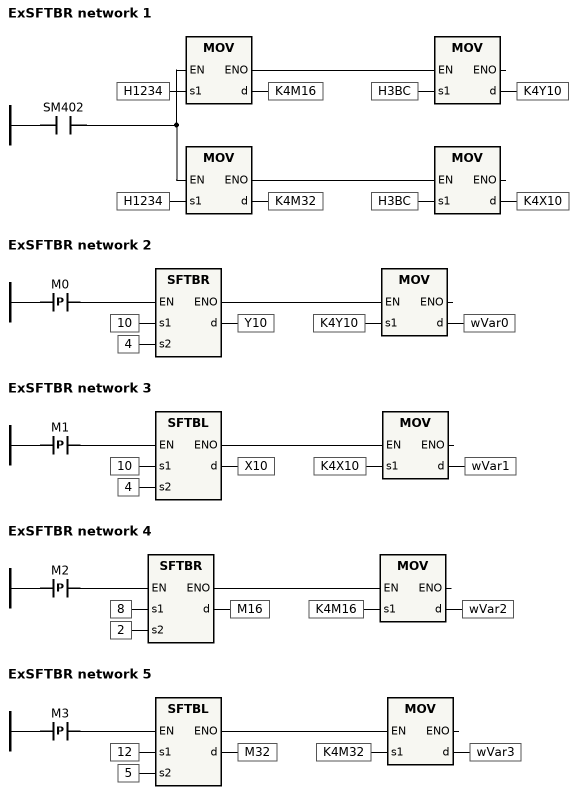
(* network 1 *)
_e1 := MOV(SM402, H1234, K4M16);
MOV(_e1, H3BC, K4Y10);
_e2 := MOV(SM402, H1234, K4M32);
MOV(_e2, H3BC, K4X10);
(* network 2 *)
_e1 := SFTBR(LDP(TRUE, M0), 10, 4, Y10);
MOV(_e1, K4Y10, wVar0);
(* network 3 *)
_e1 := SFTBL(LDP(TRUE, M1), 10, 4, X10);
MOV(_e1, K4X10, wVar1);
(* network 4 *)
_e1 := SFTBR(LDP(TRUE, M2), 8, 2, M16);
MOV(_e1, K4M16, wVar2);
(* network 5 *)
_e1 := SFTBL(LDP(TRUE, M3), 12, 5, M32);
MOV(_e1, K4M32, wVar3);
END_PROGRAM

PROGRAM ExSFTR
(* structured ladder/FBD written out as ST: instructions are called as NAME(EN, inputs, outputs); _pN, _eN, _tN stand for wires *)
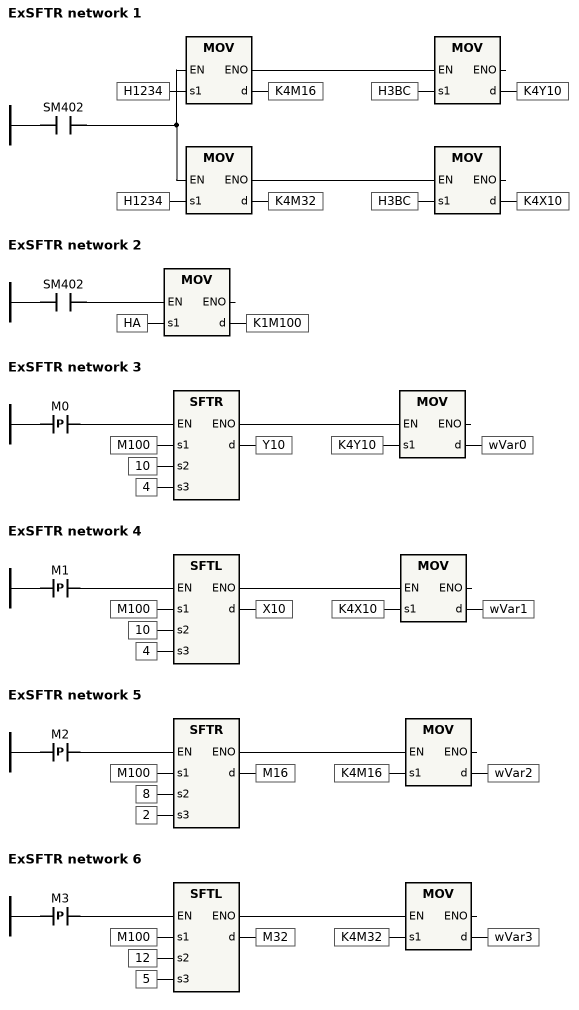
(* network 1 *)
_e1 := MOV(SM402, H1234, K4M16);
MOV(_e1, H3BC, K4Y10);
_e2 := MOV(SM402, H1234, K4M32);
MOV(_e2, H3BC, K4X10);
(* network 2 *)
MOV(SM402, HA, K1M100);
(* network 3 *)
_e1 := SFTR(LDP(TRUE, M0), M100, 10, 4, Y10);
MOV(_e1, K4Y10, wVar0);
(* network 4 *)
_e1 := SFTL(LDP(TRUE, M1), M100, 10, 4, X10);
MOV(_e1, K4X10, wVar1);
(* network 5 *)
_e1 := SFTR(LDP(TRUE, M2), M100, 8, 2, M16);
MOV(_e1, K4M16, wVar2);
(* network 6 *)
_e1 := SFTL(LDP(TRUE, M3), M100, 12, 5, M32);
MOV(_e1, K4M32, wVar3);
END_PROGRAM

PROGRAM ExSFTWR
VAR
  Mov4INT_1 : Mov4INT;
  Mov4INT_2 : Mov4INT;
  Mov8INT_1 : Mov8INT;
  Mov8INT_2 : Mov8INT;
  Mov4INT_3 : Mov4INT;
  Mov4INT_4 : Mov4INT;
  Mov4INT_5 : Mov4INT;
  Mov4INT_6 : Mov4INT;
END_VAR
(* structured ladder/FBD written out as ST: instructions are called as NAME(EN, inputs, outputs); _pN, _eN, _tN stand for wires *)
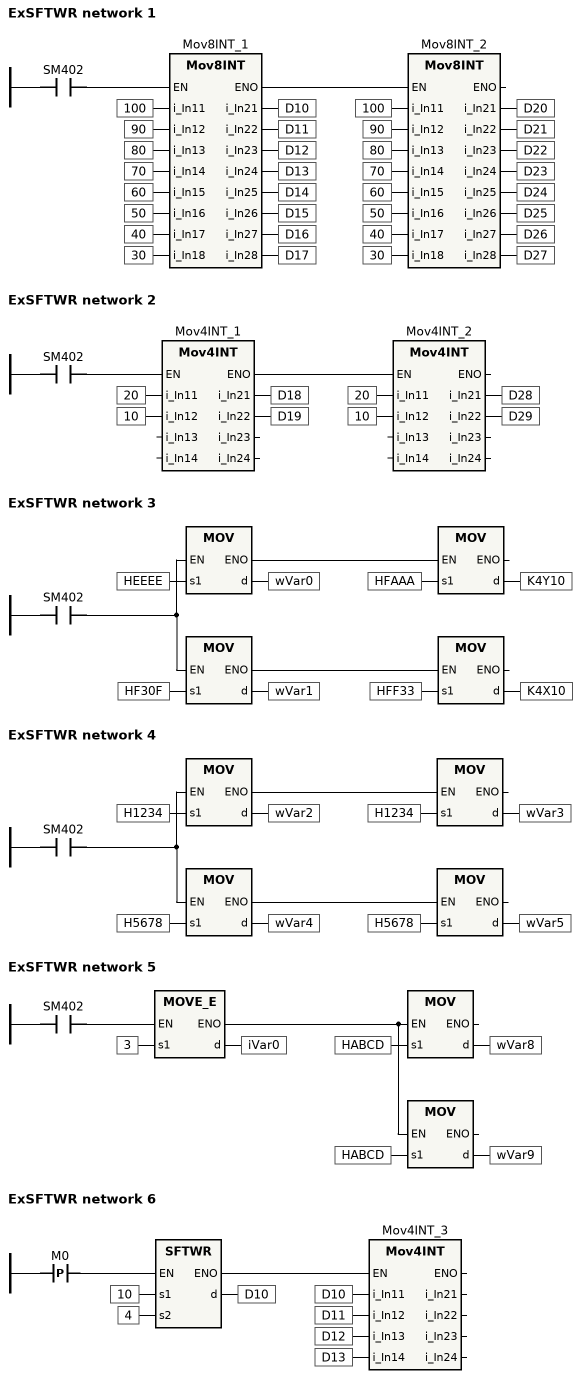
(* network 1 *)
Mov8INT_1(EN := SM402, i_In11 := 100, i_In12 := 90, i_In13 := 80, i_In14 := 70, i_In15 := 60, i_In16 := 50, i_In17 := 40, i_In18 := 30, i_In21 => D10, i_In22 => D11, i_In23 => D12, i_In24 => D13, i_In25 => D14, i_In26 => D15, i_In27 => D16, i_In28 => D17);
Mov8INT_2(EN := Mov8INT_1.ENO, i_In11 := 100, i_In12 := 90, i_In13 := 80, i_In14 := 70, i_In15 := 60, i_In16 := 50, i_In17 := 40, i_In18 := 30, i_In21 => D20, i_In22 => D21, i_In23 => D22, i_In24 => D23, i_In25 => D24, i_In26 => D25, i_In27 => D26, i_In28 => D27);
(* network 2 *)
Mov4INT_1(EN := SM402, i_In11 := 20, i_In12 := 10, i_In21 => D18, i_In22 => D19);
Mov4INT_2(EN := Mov4INT_1.ENO, i_In11 := 20, i_In12 := 10, i_In21 => D28, i_In22 => D29);
(* network 3 *)
_e1 := MOV(SM402, HEEEE, wVar0);
MOV(_e1, HFAAA, K4Y10);
_e2 := MOV(SM402, HF30F, wVar1);
MOV(_e2, HFF33, K4X10);
(* network 4 *)
_e1 := MOV(SM402, H1234, wVar2);
MOV(_e1, H1234, wVar3);
_e2 := MOV(SM402, H5678, wVar4);
MOV(_e2, H5678, wVar5);
(* network 5 *)
_e1 := MOVE_E(SM402, 3, iVar0);
MOV(_e1, HABCD, wVar8);
MOV(_e1, HABCD, wVar9);
(* network 6 *)
_e1 := SFTWR(LDP(TRUE, M0), 10, 4, D10);
Mov4INT_3(EN := _e1, i_In11 := D10, i_In12 := D11, i_In13 := D12, i_In14 := D13);
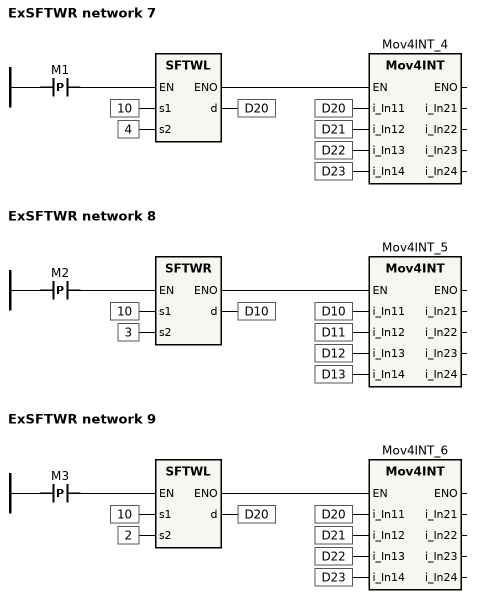
(* network 7 *)
_e1 := SFTWL(LDP(TRUE, M1), 10, 4, D20);
Mov4INT_4(EN := _e1, i_In11 := D20, i_In12 := D21, i_In13 := D22, i_In14 := D23);
(* network 8 *)
_e1 := SFTWR(LDP(TRUE, M2), 10, 3, D10);
Mov4INT_5(EN := _e1, i_In11 := D10, i_In12 := D11, i_In13 := D12, i_In14 := D13);
(* network 9 *)
_e1 := SFTWL(LDP(TRUE, M3), 10, 2, D20);
Mov4INT_6(EN := _e1, i_In11 := D20, i_In12 := D21, i_In13 := D22, i_In14 := D23);
END_PROGRAM

PROGRAM ExWSFR
VAR
  Mov4INT_7 : Mov4INT;
  Mov4INT_1 : Mov4INT;
  Mov4INT_2 : Mov4INT;
  Mov8INT_1 : Mov8INT;
  Mov8INT_2 : Mov8INT;
  Mov4INT_3 : Mov4INT;
  Mov4INT_4 : Mov4INT;
  Mov4INT_5 : Mov4INT;
  Mov4INT_6 : Mov4INT;
  Mov4INT_8 : Mov4INT;
END_VAR
(* structured ladder/FBD written out as ST: instructions are called as NAME(EN, inputs, outputs); _pN, _eN, _tN stand for wires *)
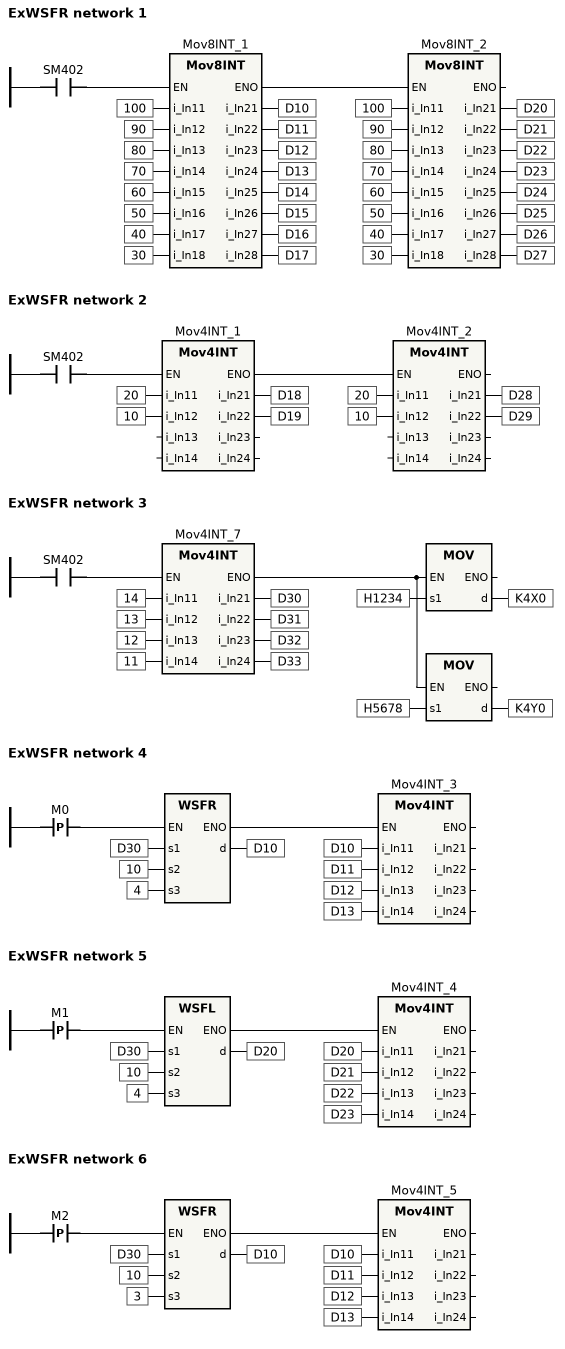
(* network 1 *)
Mov8INT_1(EN := SM402, i_In11 := 100, i_In12 := 90, i_In13 := 80, i_In14 := 70, i_In15 := 60, i_In16 := 50, i_In17 := 40, i_In18 := 30, i_In21 => D10, i_In22 => D11, i_In23 => D12, i_In24 => D13, i_In25 => D14, i_In26 => D15, i_In27 => D16, i_In28 => D17);
Mov8INT_2(EN := Mov8INT_1.ENO, i_In11 := 100, i_In12 := 90, i_In13 := 80, i_In14 := 70, i_In15 := 60, i_In16 := 50, i_In17 := 40, i_In18 := 30, i_In21 => D20, i_In22 => D21, i_In23 => D22, i_In24 => D23, i_In25 => D24, i_In26 => D25, i_In27 => D26, i_In28 => D27);
(* network 2 *)
Mov4INT_1(EN := SM402, i_In11 := 20, i_In12 := 10, i_In21 => D18, i_In22 => D19);
Mov4INT_2(EN := Mov4INT_1.ENO, i_In11 := 20, i_In12 := 10, i_In21 => D28, i_In22 => D29);
(* network 3 *)
Mov4INT_7(EN := SM402, i_In11 := 14, i_In12 := 13, i_In13 := 12, i_In14 := 11, i_In21 => D30, i_In22 => D31, i_In23 => D32, i_In24 => D33);
MOV(Mov4INT_7.ENO, H1234, K4X0);
MOV(Mov4INT_7.ENO, H5678, K4Y0);
(* network 4 *)
_e1 := WSFR(LDP(TRUE, M0), D30, 10, 4, D10);
Mov4INT_3(EN := _e1, i_In11 := D10, i_In12 := D11, i_In13 := D12, i_In14 := D13);
(* network 5 *)
_e1 := WSFL(LDP(TRUE, M1), D30, 10, 4, D20);
Mov4INT_4(EN := _e1, i_In11 := D20, i_In12 := D21, i_In13 := D22, i_In14 := D23);
(* network 6 *)
_e1 := WSFR(LDP(TRUE, M2), D30, 10, 3, D10);
Mov4INT_5(EN := _e1, i_In11 := D10, i_In12 := D11, i_In13 := D12, i_In14 := D13);
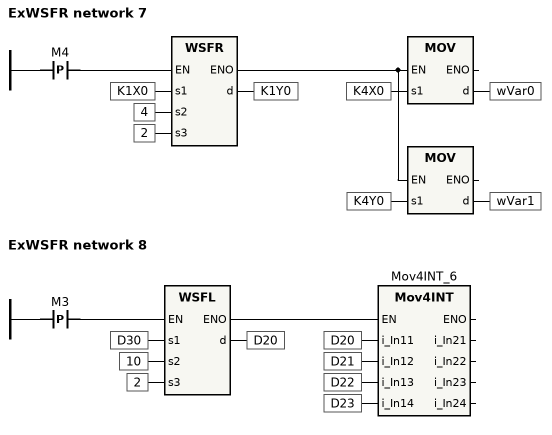
(* network 7 *)
_e1 := WSFR(LDP(TRUE, M4), K1X0, 4, 2, K1Y0);
MOV(_e1, K4X0, wVar0);
MOV(_e1, K4Y0, wVar1);
(* network 8 *)
_e1 := WSFL(LDP(TRUE, M3), D30, 10, 2, D20);
Mov4INT_6(EN := _e1, i_In11 := D20, i_In12 := D21, i_In13 := D22, i_In14 := D23);
END_PROGRAM
